# EPICS autosave request: trunk/ipApp/Db/LakeShore330_settings.req
# FILE... LakeShore330_settings.req
# USAGE.. LakeShore330.db fields to autosave.

$(P)LS330:$(Q):Gain_set.VAL
$(P)LS330:$(Q):Rset_set.VAL
$(P)LS330:$(Q):Rate_set.VAL
$(P)LS330:$(Q):RampR_set.VAL
$(P)LS330:$(Q):Ramp_on.VAL
$(P)LS330:$(Q):wr_SP.VAL
$(P)LS330:$(Q):Units_sel.VAL
$(P)LS330:$(Q):Input_sel.VAL
$(P)LS330:$(Q):HeatRg.VAL
$(P)LS330:$(Q):read.SCAN
$(P)LS330:$(Q):rd_rdat_scalc.SCAN
